(* IEC 61131-3 sources: ATCMcontrol_Engineering/src/TargetBase/Libs/ATCM_IEC1131_3/table_36, 3 files *)

(* ---- ctd.st ---- *)
(*[[
    UserURL= "ATCMfile:TOF.htm"
]]*)
(*
 *  IEC-1131-3 Standard Functionblock CTD for data type INT
 *  Purpose: Down Counter
 *)
FUNCTION_BLOCK CTD
VAR_INPUT  (* Inputs *)
    CD         : BOOL R_EDGE; (* count down if rising edge     *)
    LD         : BOOL;        (* if true, copy PV to CV        *)
    PV         : INT;         (* start value                   *)
END_VAR
VAR_OUTPUT (* Outputs *)
    Q          : BOOL;        (* TRUE if CV <= 0               *)
    CV         : INT;         (* counter output                *)
END_VAR

inline { STDLIB(ctd) }

END_FUNCTION_BLOCK

(* ---- ctu.st ---- *)
(*[[
    UserURL= "ATCMfile:TON.htm"
]]*)
(*
 *  IEC-1131-3 Standard Functionblock CTU for data type INT
 *  Purpose: Up Counter
 *)
FUNCTION_BLOCK CTU
VAR_INPUT (* Inputs *)
    CU         : BOOL R_EDGE; (* count up if rising edge *)
    R          : BOOL;        (* if true,  CV to zero    *)
    PV         : INT;         (* end value               *)
END_VAR
VAR_OUTPUT (* Outputs *)
    Q          : BOOL;        (* TRUE if CV >= PV        *)
    CV         : INT;         (* counter output          *)
END_VAR

inline { STDLIB(ctu) }

END_FUNCTION_BLOCK

(* ---- ctud.st ---- *)
(*[[
    UserURL= "ATCMfile:TP.htm"
]]*)
(*
 *  IEC-1131-3 Standard Functionblock CTUD for data type DINT
 *  Purpose: Up/Down Counter
 *)
FUNCTION_BLOCK CTUD
VAR_INPUT (* Inputs *)
    CU         : BOOL R_EDGE; (* count up if rising edge   *)
    CD         : BOOL R_EDGE; (* count down if rising edge *)
    R          : BOOL;        (* Reset, set CV to 0        *)
    LD         : BOOL;        (* if true, copy PV to CV    *)
    PV         : INT;         (* start value               *)
END_VAR
VAR_OUTPUT (* Outputs *)
    QU         : BOOL;        (* TRUE if CV >= PV          *)
    QD         : BOOL;        (* TRUE if CV <= 0           *)
    CV         : INT;         (* counter output            *)
END_VAR

inline { STDLIB(ctud) }

END_FUNCTION_BLOCK
